// TIA Portal V16 export
// export: Created 2021-11-12T13:32:41.4627702Z, ExportSetting WithDefaults, DisplayName Totally Integrated Automation Portal, DisplayVersion V16 Update 3, DisplayName TIA Portal Version Control Interface, DisplayVersion V16 Update 2, DisplayName TIA Portal Openness, DisplayVersion V16 Update 3, DisplayName SINAMICS Startdrive Advanced, DisplayVersion V16 Update 5, DisplayName SINAMICS Startdrive G130, G150, S120, S150, SINAMICS MV, S210, DisplayVersion V16 Update 5, DisplayName SINAMICS Startdrive G110M, G120, G120C, G120D, G120P, G115D, DisplayVersion V16 Update 5, DisplayName STEP 7 Professional, DisplayVersion V16 Update 3, DisplayName STEP 7 Safety, DisplayVersion V16, DisplayName WinCC UA Professional, DisplayVersion V16 Update 3
DATA_BLOCK "STATUS_200+UH11"   // DB57
{ S7_Optimized_Access := 'TRUE' }
VERSION : 0.1
// stored: AutoNumber true, DBAccessibleFromOPCUA true, IsOnlyStoredInLoadMemory false, IsRetainMemResEnabled false, IsWriteProtectedInAS false, MemoryReserve 100
   VAR
      xxxxx___BinarySensors___xxxxx : Byte;
      xxxxx___BinaryOthers___xxxxx : Byte;
      SF02_14 : Bool;   // Start automat
      SF03_14 : Bool;   // Nulování poruchy
      SF04_14 : Bool;   // Reset bezpečnostního okruhu
      SF05_22 : Bool;   // Blokování pásu v peci 3
      SF06_22 : Bool;   // Blokování pásu v peci 1
      SF07_22 : Bool;   // Blokování pásu v peci 2
      "I450.6" : Bool;   // Rezerva
      "I450.7" : Bool;   // Rezerva Okamžitý stop Robot 2R3
      "I451.0" : Bool;   // Rezerva Okamžitý stop Robot 2R4
      "I451.1" : Bool;   // Rezerva Okamžitý stop Robot 2R5
      "I451.2" : Bool;   // Rezerva Okamžitý stop Robot 2R6
      "UF01-SF02_14" : Bool;   // Bedna Žádost o výměnu
      "UF01-SF03_14" : Bool;   // Bedna Vyměněna
      "I451.5" : Bool;   // Rezerva Vzorek na test
      "I451.6" : Bool;   // Rezerva Materiál vložit
      "I451.7" : Bool;   // Rezerva
      xxxxx___InterfaceSignals___xxxxx : Byte;
      SumErr : Bool;   // Sum of significant errors
      PwrOK : Bool;   // Significant switches ON
      xxxxx___AnalogueSensors___xxxxx : Byte;
      xxxxx___Drives___xxxxx : Byte;
      xxxxx___Other___xxxxx : Byte;
      xxxxx___Alarms___xxxxx : Byte;
      ES : Struct   // E-stop
         Main { S7_SetPoint := 'True'} : "UDT_Status_main";
         Specific { S7_SetPoint := 'True'} : "UDT_DI_Mon_Status_specific";
         Error { S7_SetPoint := 'True'} : "UDT_Error01";
      END_STRUCT;
      KF31 : Struct   // module 200UH11- KF31
         Main { S7_SetPoint := 'True'} : "UDT_Status_main";
         Specific { S7_SetPoint := 'True'} : "UDT_DI_Mon_Status_specific";
         Error { S7_SetPoint := 'True'} : "UDT_Error01";
      END_STRUCT;
   END_VAR
BEGIN
END_DATA_BLOCK
